(* IEC 61131-3 sources: Dev/Dev_V200/200 (part 4) *)

	   _229_S : UDINT := SIZEOF(NH_FRM_229); _229 : NH_FRM_229;
   	_230_S : UDINT := SIZEOF(NH_FRM_230); _230 : NH_FRM_230;
	   _231_S : UDINT := SIZEOF(NH_FRM_231); _231 : NH_FRM_231;
		_232_S : UDINT :=	SIZEOF(NH_FRM_232); _232 : NH_FRM_232;
		_233_S : UDINT :=	SIZEOF(NH_FRM_233); _233 : NH_FRM_233;
		_234_S : UDINT :=	SIZEOF(NH_FRM_234); _234 : NH_FRM_234;
		_235_S : UDINT :=	SIZEOF(NH_FRM_235); _235 : NH_FRM_235;
		_236_S : UDINT :=	SIZEOF(NH_FRM_236); _236 : NH_FRM_236;

		_246_S : UDINT :=	SIZEOF(NH_FRM_246); _246 : NH_FRM_246;
	//	_247_S : UDINT :=	SIZEOF(NH_FRM_247); _247 : NH_FRM_247;
		_248_S : UDINT :=	SIZEOF(NH_FRM_248); _248 : NH_FRM_248;
	//	_249_S : UDINT :=	SIZEOF(NH_FRM_249); _249 : NH_FRM_249;
		_260_S : UDINT := SIZEOF(NH_FRM_260); _260 : NH_FRM_260 ;

(*
   _0_S : UDINT := SIZEOF(NH_FRM_0); _0 : NH_FRM_0 ;
   _0_S : UDINT := SIZEOF(NH_FRM_0); _0 : NH_FRM_0 ;
   _0_S : UDINT := SIZEOF(NH_FRM_0); _0 : NH_FRM_0 ;
*)

	   _END_FRM_WEB    : UDINT := 0;

	END_VAR

	FUNCTION_BLOCK _Nh_Create_FRM
   	VAR_INPUT
         Go          : USINT;
			all			: BOOL;
   	END_VAR
   	VAR_OUTPUT
         done        : BOOL;
			busy			: BOOL;
	      cyc         : UINT;
   	   files       : UINT;
      	actSize     : UDINT;
//         expTime    	: TIME;
   		GoNext		: USINT;
		END_VAR
   	done  := false;
      CASE go OF
       0 :  RETURN;
       1 :
            xFrmHed  := ADR(_START_FRM_SYS);
            Go 		:= 3;
				IF all THEN
					_Nh_Log_Path(wh:=21, frm:=1);
// 	           rb       := ForceDirs(fileName := yTx2);
					yTx2 		:= CONCAT('New FRM_SYS: ',yTx2);
 					rb 		:= _Nh1RowTxt(logRst := 1);
					GoNext   := 2;
   			ELSE
					GoNext   := 0;
				END_IF;
				all	:= false;
       2 :
      		GoNext	:= 0;
				{$IFDEF __NH_WEB}
					xFrmHed  := ADR(_START_FRM_WEB);
					_Nh_Log_Path(wh:=21, frm:=1);
					yTx2 		:= CONCAT('New FRM_WEB: ',yTx2);
 					rb 		:= _Nh1RowTxt(logRst := 1);

               Go    	:= 3;
            {$ELSE}
               Go    	:= 99;
   			{$END_IF}

       3 :
				busy		:= true;
            cyc      := 0;
            files    := 0;
            actSize  := 0;
            xFrmHed  := xFrmHed + 1;
            Go       := 4;

       4 :
      	   cyc   := cyc + 1;
				_Nh_Log_Path(wh:=21, frm:=1);
            WHILE xFrmHed^.Size > 0 DO
      	      yTx3 := CONCAT(yTx2, xFrmHed^.hed.Name ,'.FRM');
         	   fH   := FileOpen(fileName := yTx3, mode := F_WRITE);
            	IF fH <> INVALID_HANDLE_VALUE THEN
               	sz       := PTR_TO_UDINT(xFrmHed) + 4;
      	         sz       := FileWrite (hFile := fH, adrBuf := sz, size := xFrmHed^.size);
         	      actSize  := actSize + sz;
            	   files    := files + 1;
               	aSys.RWtoFileCycle := aSys.RWtoFileCycle + sz;
      	      END_IF;
         	   rb       := FileClose (hFile := fH);
      	      sz       := xFrmHed^.size + 4;
         	   xFrmHed  := xFrmHed + sz;
					IF _NhMaxRWLimit() OR _NhMaxTimeCyc()  THEN
						EXIT;
					END_IF;
(*
      	      expTime  := SUB_DT_DT(GetRTC(),aSys.NhDT);
      	      IF aSys.RWtoFileCycle > 32768 OR expTime > T#0.2s THEN
         	      EXIT;
            	END_IF;
*)
      	   END_WHILE;
         	IF xFrmHed^.Size = 0 THEN
               Go       := 99;
      	   END_IF;
       99:
				Go := GoNext;
				IF Go = 0 THEN
         	   Done := TRUE;
         	   Busy := false;
				END_IF;
      END_CASE;
	END_FUNCTION_BLOCK

	VAR_GLOBAL
   	fb_Nh_Create_FRM    : _Nh_Create_FRM;
	END_VAR

{ $ END_IF }

(* ---- _Nh_Het.st ---- *)
TYPE

(*
   NH_HET_DIS	{HIDDEN} :  STRUCT 		    // prenos medzi HET a TGL,WSB....
		ok 			: BOOL;                 	// mame ReQ teplotu z tohto regulatora
		chg			: BOOL;       				   // zmena ReQ
		valReQ		: REAL;                    // pozadovana velicina
		valAct		: REAL;                    // aktualna velicina
   END_STRUCT;
*)

END_TYPE

TYPE

END_TYPE

TYPE
END_TYPE

TYPE
END_TYPE

FUNCTION _Nh_PvValOut  {HIDDEN} : USINT		// nastavi vystupny stupen KURENIA/CHLADENIA podla hysterezie
	VAR_INPUT
   	het		: BOOL;
		up			: USINT;
		pv			: USINT;
		reQ		: REAL;
		val		: REAL;
		wht		: PTR_TO NH_HET_MODE;
  	END_VAR
//	vr	:= wht^.reQ[ pv ];
	i	:= 3;
	WHILE i >= 1 DO
		kr := wht^.hys[up,i];

(*
		IF up THEN
			kr		:= wht^.hys.up[i];
		ELSE
			kr		:= wht^.hys.dn[i];
		END_IF;
*)
		IF het THEN														// kurenie

(*
					UP                 		DN
			23.3  0.                      0.
			23.2  0.                      0.
			23.1  0.                 		1.	<= [23+0.1=23.1]
			23.0  0 --------------------- 1.
			22.9	0.                      2.	<= [23-0.1=22.9]
			22.8  0.                      2.
			22.7  0.                      2.
			22.6	0.	                     2.
			22.5  1.	<= [23-0.5=22.5]     2.
			22.4  1.                      2.
			22.3  1.                      3.	<= [23-0.7=22.3]
			22.2  1.                      3.
			22.1  1.                      3.
			22.0  2.	<= [23-1.0=22.0]     3.
			21.9  2.                      3.
			21.8  2.                      3.
			21.7  2.
			21.6  2.
			21.5  2.
			21.4  2.
			21.3  2.
			21.2  2.
			21.1  2.
			21.0  3.	<= [23-2.0=21.0]
			20.9	3.
*)

//			IF val <= reQ - kr THEN
			IF val <= reQ + kr THEN
				EXIT;
			END_IF;
		ELSIF	pv = 0 THEN												// pri chladenie/vetrani/odvlhceni je PV=0 OFF
			i := 1;
		ELSIF val >= reQ + kr THEN
			EXIT;
		END_IF;
		i := i-1;
	END_WHILE;
	_Nh_PvValOut := i;
END_FUNCTION

TYPE

END_TYPE

(* ---- _Nh_Ini.st ---- *)
(* INICIALIZACNE FUNKCIE RAM A DBX PO RESTARTE, OBNOVENIE Z SDC A TESTY KONZISTENCIE  *)
(*
TYPE
  	NH_DBX_2	{HIDDEN}   :  STRUCT 			// riadiaca hlavicka DBX
      ver         : NH_DBX_VER   ;
      sCfg        : USINT := SIZEOF(NH_CFG_CFG);       // velkost vety aCfg v DBX
      sPar        : USINT := SIZEOF(NH_PAR_CFG);       // velkost vety aPar v DBX
      sVaz        : USINT := SIZEOF(NH_VAZ_CFG);       // velkost vety aVaz v DBX

      nCfg        : USINT := _Nh_CFG;              // pocet viet CFG
      nPar        : USINT := _Nh_PAR;              // pocet viet PAR
      nVio        : USINT := _Nh_VAZ;              // pocet viet VAZ
      // adresy dat
      aCfg        : UINT;                          // offset od _Dbx0  - zaciatok aCfg ulozeny v databoxe
      aPar        : UINT;                          // zaciatok aPar ulozeny v databoxe
      aVio        : UINT;                          // zaciatok aVaz ulozeny v databoxe
      vRam        : UINT;                          // aktualna velkost dat v aRam[] = posladny zaznam aVaz
      // gobalne  premenne/sablony, ktore sa obnovuju z DBX
      all         : NH_DBX_VAR;
      rezerva     : STRING[79];
//    0,ROM,ZON,CAT,SCN,FAV,USR,HET,SVD,SVA,RGB,ZAS,STY,VEN,ROL,GAR,SIR,13,WSB,TLA,KOT,TVE,CER,PIR,TER,DOR,WIN,LUX,KEY,H20,FIR,GAS,
//      ixc         : ARRAY[0..50] OF USINT := [0,3,1,2,5,4,20,22,6,10,11,12,21,23,31,32,30,13,14,8,7,9,15,16,17,18,19,24,27,28,29,38,39,0]; // SCN,SVD,SVA....
//      ixc         : ARRAY[0..50] OF USINT := [0,1,3,4,5,20,22,10,11,12,21,23,31,32,33,34,35,30,13,14,24,15,19,16,17,18,6,7,8,9,27,28,29,37,38,39,2,0]; // SCN,SVD,SVA....
	END_STRUCT;

   NH_CFG_CFG_2  {HIDDEN}:  STRUCT 					// zakladny konfiguracny subor vsetkych DEV a ich rozlozenie v RAM
      // spoloxna struktura pre xNh
		Siz         : UDINT;								// velkost jedneho zaznamu
		Ram         : UDINT;							  // adresa 1.vety vo virtualnej pamati mRam[ vRam ], kde je ulozena xCfg (nulta veta )
      Rec         : INT;                       // pocet zaznamov
		New			: INT;						     // pocet novych zanamov, ktore sa ziadaju
      nDe         : USINT;                       // pocet DEL-viet
      rDe         : INT;                       // posledna volna DEL veta
      NOk         : BOOL;                      // novopridana veta bude oznacena uz pri pridani ako platna
      ver         : USINT := 1;
		// dotial musia mut CFG,PAR,VAZ rovnake, kebo sa pouzivaju xNh^
  		cfg			: STRING[3] ;						// nazov suboru na SDC dev := xxx.***
      ofs         : UDINT;                       // offset Empty premennej od eRom
      // unikatne  pre CFG
      par         : USINT;                      // cislo parametra  (odkaz do aPar)
      al          : USINT;	// := SIZEOF(NH_DEV_ALL) ;                      // velkost specialnej cfg pre dev
      cx          : USINT;                      // velkost specialnej cfg pre dev
      // dotialto sa obnovuje DBXver=001
      cf          : USINT := SIZEOF(NH_CFG_ALL);                      // velkost hlavnej cfg
      me          : UINT;                       // velkost uzivatelskej prevadzkovej pamate
      hw          : USINT;                       // velkost HW pamate
      io      		: USINT;
      dummy5      : USINT;
      dummy6      : USINT;
      dummy7      : USINT;
      dummy8      : USINT;
      dummy9      : USINT;
      // dotialto sa obnovuje DBXver > 001
      cat         : USINT;                      // cislo cat do ktorej patri toto dev
      ref         : USINT := 251;               // druh refreshu 251-len to co je na obrazovke,252=to co je na obrazevke a predefinovat,254=novy vypis od 1.zanamu
//      cou         : USINT;                      // cislo skupiny vystupov pre prenos vstupov
      tgr         : USINT;                      // typovy predstavitel/skupina vazieb

      mna         : USINT;                      // cislo menu pre ikonu vlastnosti - administrator _042.MN0
      mnu         : USINT;                      // cislo menu pre ikonu vlastnosti - user          _042.MN0
      rExp        : USINT;                      // pocet viet v z exportu
      fBr         : USINT;                      // cislo formatoveho suboru pre pre BRW-ROW, ulozene _Nh_ADR_ROT,'/CFG/FRM/_000.
      fSc         : USINT := 200;               // cislo menu cez ktore sa dostane so _Nh_Frm_SCR = parametrov DEV
      ar2         : BOOL;                       // '>>' dvojita      sipka dalej je v obr[4] prioritou c.1
      lst         : BOOL;                       // ma ikonu DEV-listu {SCN,ACT..}
      stp         : BOOL := true;               // moze mat odskok na vazby = ikona setup (len v rezime setup)
      fav         : BOOL := true;               // ma ikonu fav
      chk         : BOOL := true;               // ma ikonu check (ak je vo vazbach)
      edn         : BOOL := true;               // moze sa editovat nazov
      sld         : BOOL;                       // DEv ma slider v riadkovom zobrazeni
      ou          : BOOL;                       // tot je vystup - kde sa nieco nastavuje
      dbx         : BOOL;                       // data boli obnovene z DBX
      sdc         : BOOL;                       // data boli obnovene z SDC
//      NoDelDBX    : BOOL;                       // pri obnoveni z DBX sa NE-oznaci ako DEL. Potom ju odznaci proces aktualizacie adries z NH2.ADR
      NoRecCat    : BOOL;                       // pri zfiltrovani kategorie sa zobrazia aj ked nemaju ziadny zaznam
      AllCFG      : BOOL;                       // z DBX neobnovuje po cf+al+cx... ale obnovi naraz cely zaznam podls velkosti SIZE
      scn         : BOOL;                       // priznak, ze ide o dev, ktore riadi viac vystupnych DEV (SCN,ACT,TIM...)  ma nejeky dev-list
      body        : BOOL;                       // tento DEV zapisuje pritomnost
      ini         : BOOL;                       // pri inicializacii boli pridane vety, treba ich popisat
      del         : BOOL;			               // je mozne mazat DEV (ON/OFF)
      bck         : BOOL := true;               // toto cfg sa zalohuje z RAM -> SDC
      imp         : BOOL := true;               // do cf sa importuju adresy  z CIB .... , ROM nebude mat adresy
      NewExp      : BOOL;                       // toto CFG ma z exportu nove data/adresy a musi sa aktualizovat
      QckStat     : BOOL;                       // v HOME-QuickMnu sa vypisuju obrazku zo stat, nie z dev
      lvl254      : BOOL;                       // dev nema max LVL 100% ale 254 = DALI            (len pre web)
      analog      : BOOL;                       // dev je 0-100% alebo 0-254                       (len pre web)
      dali      	: BOOL;                       // patri do dali
      ShwSta   	: BOOL;  		              // robrazi sa ikona cfg v ROM/ZON ak je niektore z DEV v [cf] aktivne
      zone        : BOOL;                       // moze vstupovat {davat signal} aj do zony  (TER,LUX)

   END_STRUCT;

  	NH_PAR_CFG_2  {HIDDEN}:  STRUCT 					// zakladny konfiguracny subor vsetkych parametrov
      // spoloxna struktura pre xNh
		Siz         : UDINT;								// velkost jedneho zaznamu
		Ram         : UDINT;							  // adresa 1.vety vo virtualnej pamati mRam[ vRam ], kde je ulozena xCfg (nulta veta )
      Rec         : INT;                       // pocet zaznamov
		New			: INT;						     // pocet novych zanamov, ktore sa ziadaju
      nDe         : USINT;                       // pocet DEL-viet
      rDe         : INT;                       // posledna volna DEL veta
      NOk         : BOOL;                      // novopridana veta bude oznacena uz pri pridani ako platna
      ver         : USINT := 1;

		cfg			: STRING[3] ;						// nazov suboru na SDC dev := xxx.***
      ofs         : UINT;                       // offset Empty premennej od epSvd

      // unikatne  pre PAR
      dbx         : BOOL;                       // data boli obnovene z DBX
      sdc         : BOOL;                       // data boli obnovene z SDC
//		in          : BOOL := true;					//	vo vazbe IN sa vytvara parameter, inak sa preberie z hlavicky
//		ou          : BOOL := true;					// vo vazbe OU sa vytvara parameter, inak sa preberie z hlavicky
      grp         : BOOL;                       // novy parameter sa vytvori, len ak vstupuje na pozici OUT skupinovych prikazov do SCN,ACT,TIM. Inak sa zoberie default cislo paramtra z DEV
//		New			: INT;						     // pocet novych zanamov, ktore sa ziadaju
	END_STRUCT;

  	NH_VIO_CFG_2	{HIDDEN}   :  STRUCT 			  // zakladny konfiguracny subor vazieb
		Siz         : UDINT := SIZEOF(NH_VAZ);	  // velkost jedneho zaznamu
		Ram         : UDINT;							  // adresa 1.vety vo virtualnej pamati mRam[ vRam ], kde je ulozena xCfg (nulta veta )
      Rec         : INT;                       // pocet zaznamov
		New			: INT;						     // pocet novych zanamov, ktore sa ziadaju
      nDe         : USINT;                       // pocet DEL-viet
      rDe         : INT;                       // posledna volna DEL veta
      NOk         : BOOL;                      // novopridana veta bude oznacena uz pri pridani ako platna
      ver         : USINT := 1;

      ref         : BOOL := true;              // vsetky vazby sa refreshnu (ako keby bolo cmd > 0)
	   ini         : BOOL;                      // pri restarte sa nplni DEFAULT hodnotami
   END_STRUCT;
END_TYPE

VAR_GLOBAL
	oDbx	      {HIDDEN}	   : NH_DBX_2;                                // hlavny riadiaci subor vratane organizacie DBX
   oCfg        {HIDDEN}    : NH_CFG_CFG_2;                            // konfiguracia vsetkych DEV
   oPar        {HIDDEN}    : NH_PAR_CFG_2;                            // konfiguracia vsetkych DEV
   oVio        {HIDDEN}    : NH_VIO_CFG_2;                            // konfiguracia vsetkych DEV
END_VAR
*)

VAR_GLOBAL CONSTANT
(*
  _NhQickGuide   {HIDDEN} : ARRAY[ 9..16,0..1] OF USINT :=
                    [   1,  0,                     // Vytvorit miestnost
                        2, 44,                     // Dev bezmiestnosti
                        2, 16,
                        2, 15,
                        2, 24,
                        2, 14,
                        2,  5,
                        2,  6
                    ];
END_VAR
*)

  _NhQickGuide   {HIDDEN} : ARRAY[ 9..14,0..1] OF USINT :=
                    [   2, 16,
                        2, 15,
                        2, 24,
                        2, 14,
                        2,  5,
                        2,  6
                    ];
END_VAR

FUNCTION _NhNewPAR {HIDDEN} : BOOL	    // zvysi poziadavku na novu vetu (vrati true), alebo oznaci existujucu ak je DEL (false)
   VAR_INPUT
      xP    : PTR_TO INT;                          // xCfg^.par, alebo io.p
      cp    : USINT;
		ee	: INT;
   END_VAR
   _NhNewPAR := true;                             // default nepridavaju sa nove vety

(*
	IF cp = 14 THEN
      yTx2     := CONCAT('  nd: ',INT_TO_STRING(nd), ' cp: ',USINT_TO_STRING(cp),' np: ',INT_TO_STRING(xP^)   );
      _Nh1RowTxt(logRst:=1, noTime := 1);

//		aSys.ini := 217;
//		RETURN;

	END_IF;
*)

   IF xP^ = 0	THEN																// nememe parameter a mal by byt
      ;
   ELSIF xP^ > aPar[cp].rec THEN                   // parameter sa este len prida, ale uz si ho nieco rezervovalo
		j := j+1;
	ELSIF _NhxPar(cp := cp, np := xP^ ,x:=ee) THEN   // uz si ho zobralo iny DEV, musi sa vytvoriy novy
		i := i + 1;
   ELSE
       _NhNewPAR   := false;                        // pridava sanew := true;
       xPar^.ok.ok := true;
		z := z + 1;
   END_IF;
   IF _NhNewPAR THEN
      aPar[cp].new   := aPar[cp].new + 1;
      aPar[cp].nOk   := true;                                        // pridane vety budu hned platne
      xP^            := aPar[cp].rec + aPar[cp].new;   // parametrom bude nova platna veta
		x				 	:= x + 1;
   END_IF;
(*
	IF cp = 14 THEN
      yTx2     := CONCAT('    j: ',SINT_TO_STRING(j), ' i:',USINT_TO_STRING(i), ' z:',INT_TO_STRING(z),' x:',INT_TO_STRING(x)   );
      _Nh1RowTxt(logRst:=1, noTime := 1);
	END_IF;
*)

END_FUNCTION

FUNCTION _Nh_Ini_PAR_Test {HIDDEN}   : BOOL	    // prejde vsetky DEV, ktore maju parametre a tieto parametre prida,a lebo od-DELETUJE
   VAR_TEMP
      cp       : USINT;
   END_VAR
   IF aSys.exp = 0 THEN
      yTx2     := 'START - _Nh_Ini_PAR_Test KONTROLA PARAMETROV :';
      _Nh1RowTxt(logRst:=1);
   END_IF;
   aSys.exp := aSys.exp + 1;
   WHILE aSys.exp <= aDbx.nCfx[0] DO                                       // prechadzaju sa typy parametrov kazdom cykle
      IF aCfg[aSys.exp].par = 0  THEN                                          // nema cf typ CFG_ALL, a tym ani parametre
         RETURN;
      END_IF;

	x	:= 0;
	y	:= 0;
	z	:= 0;
	i	:= 0;
	j	:= 0;

      cp    := aCfg[aSys.exp].par;
      FOR nd := 1 TO aCfg[ aSys.exp ].rec DO                         // prechadza len toto cfg
			IF _NhxPt( c := aSys.exp, n := nd, x:=70) OR aCfg[aSys.exp].dali THEN           // testuje len platne vety,
				IF cp = 0 THEN
               IF xPt^.cf.par > 0 THEN
						xPt^.cf.par	:= 0;                                    // grp je len pre ACT,SCN
						y				:= y + 1;
					END_IF;
				ELSE
				   _NhNewPAR(cp := cp, xP := ADR(xPt^.cf.par), ee:=60);
				END_IF;
			END_IF;
    	END_FOR;
     	yTx2	:= '  ' +USINT_TO_STRINGF(aSys.exp,'%3d')
		  			+ ' ' + aCfg[ aSys.exp ].cfg
					+ ' Rec: ' + INT_TO_STRINGF(aCfg[aSys.exp].rec,'%3d')
					+ ' Del: ' + INT_TO_STRINGF(y,'%3d');

		IF cp > 0 THEN
	     	yTx2	:= yTx2
						+ ' Ok: '  + INT_TO_STRINGF(z,'%3d')
						+ ' New: ' + INT_TO_STRINGF(x,'%3d')
		  				+ ' ' + aPar[cp].cfg
						+ ' ' + INT_TO_STRINGF(aPar[cp].rec,'%3d')
						+ ' D: ' + USINT_TO_STRINGF(i,'%3d');
		END_IF;
		IF aCfg[ aSys.exp ].cfg <> '' THEN
	  		rb       := _Nh1RowTxt(logRst := 1);
		END_IF;
		IF x > 0 THEN
			_Nh_Go_DbxToMem(ram := true,dbx := false );                        // zalozi RAM->DBX, z DBX vrati do RAM s pridanim novych uz platnych viet
		END_IF;

      RETURN;
   END_WHILE;
   aSys.ini := 214;
   yTx2     := CONCAT('END - Kontola PAR Ok. aSys.ini:=', USINT_TO_STRING(aSys.ini) );
   rb       := _Nh1RowTxt(logRst := 1);
END_FUNCTION

FUNCTION _NhIniVAZ  {HIDDEN} : BOOL	    // prejde vazby a ak v IN alebo OUT je DEV, ktore neexistuje, vymaze vazbu
   VAR
      nvz    : USINT;
//      io    : USINT;
//      chg   : INT;
//      old   : INT;
      par   : INT;
      ndv   : INT;
      cp       : USINT;
   END_VAR
	yTx2     := '_NhIniVAZ     : ZACINAM KONTROLU';
 	_Nh1RowTxt(logRst:=1);

	FOR nvz := 2 TO 4 DO
		x	:= 0;
		y	:= 0;
		z	:= 0;
		i	:= 0;
		FOR ndv := 1 TO aVaz[nvz].Rec DO
         IF _NhxVaz( cv := nvz, nd := ndv) THEN                             // veta vazby je platna
				ok	:= true;

		  		IF _NhxPt(c:=xVaz^.in.c,n:=xVaz^.in.n,err:=1 ,x:=22) = false THEN
					xVaz^.ok.ok 	:= false;
					ok	   			:= false;
				ELSIF _NhxPt(c:=xVaz^.ou.c,n:=xVaz^.ou.n, err:=1 ,x:=24) = false THEN
					xVaz^.ok.ok 	:= false;
					ok	   			:= false;
				END_IF;

				IF ok THEN
					cp := aCfg[xVaz^.in.c].par;
					IF nvz = 3 THEN
						cp := 0;
					END_IF;
					IF cp = 0 THEN
						IF xVaz^.in.p > 0 THEN
							xVaz^.in.p := 0;
							y			  := y + 1;
						END_IF;
					ELSIF xVaz^.in.p > 0 THEN
					   _NhNewPAR(cp := cp, xP := ADR(xVaz^.in.p), ee:=61);
					END_IF;
					cp := aCfg[xVaz^.OU.c].par;
					IF cp = 0 THEN
							IF xVaz^.OU.p > 0 THEN
							xVaz^.OU.p := 0;
							y			  := y + 1;
						END_IF;
					ELSIF xVaz^.OU.p > 0 THEN
				   	_NhNewPAR(cp := cp, xP := ADR(xVaz^.OU.p), ee:=62);
					END_IF;
	         END_IF;
			END_IF;
      END_FOR;
     	yTx2	:= '   ' + USINT_TO_STRING(nvz)
		  			+ ': Rec: ' + INT_TO_STRINGF(aVaz[nvz].rec,'%3d')
					+ ' Del: ' + INT_TO_STRINGF(y,'%3d')
					+ ' Ok: '  + INT_TO_STRINGF(z,'%3d')
					+ ' New: ' + INT_TO_STRINGF(x,'%3d')
					+ ' Dupl: ' + USINT_TO_STRINGF(i,'%3d');
 		rb       := _Nh1RowTxt(logRst := 1);
		IF x > 0 THEN
			_Nh_Go_DbxToMem(RAM := true,dbx := false );                        // zalozi RAM->DBX, z DBX vrati do RAM s pridanim novych uz platnych viet
		END_IF;
	END_FOR;

	yTx2     := '_NhIniVAZ     : KONTROLA OK.';
 	_Nh1RowTxt(logRst:=1);

END_FUNCTION

FUNCTION _Nh_Ini_Default_CFG_INI {HIDDEN}    : BOOL	    // doplni default CFG, ak este nie je
	VAR_INPUT
		vz		: BOOL;
		ver	: BOOL := true;
		nOk	: BOOL := true;
		rec	: INT;
		cf		: USINT;
	END_VAR
   _Nh_Ini_Default_CFG_INI := false;                             // default nepridavaju sa nove vety
	IF vz	THEN
	   IF aVaz[cf].rec < rec  THEN   // ver=0: FAV,USR
   	   IF aVaz[cf].rec < rec THEN
      	   aVaz[cf].new :=  rec  - aVaz[cf].rec ;
	      END_IF;
   	   aVaz[cf].ini := TRUE;
      	aVaz[cf].nOk := nOk;
   	END_IF;
	 	aCfg[cf].ini   := aVaz[cf].ini OR ver;
	ELSE
		IF rec > aCfg[cf].rec THEN                                         // porovna sa aktulny pocet s pozadovanym
 			aCfg[cf].nOk	:= nOk;
	      aCfg[cf].new   := rec  - aCfg[cf].rec ;
   	   aCfg[cf].ini   := true;                                        // do tohto CFG sa budu pridavat detault vety
   		yTx2 := CONCAT('..',aCfg[cf].cfg,' + ',INT_TO_STRING(aCfg[cf].new) );
			rb   := _Nh1RowTxt(logRst := 1);
		END_IF;
		IF ver AND aCfg[cf].ver = 0 THEN
		 	aCfg[cf].ini   := true;
		END_IF;
	END_IF;
END_FUNCTION

FUNCTION _Nh_Ini_Default_CFG_DEF {HIDDEN} : BOOL	    // nakopiruje default sablony
	VAR_INPUT
		cf		: USINT;
		frm	: UINT;
	END_VAR
   _Nh_Ini_Default_CFG_DEF := false;                             // default nepridavaju sa nove vety
	IF aCfg[cf].ini = false THEN                                         // porovna sa aktulny pocet s pozadovanym
		RETURN;
	END_IF;
	// cele preddefinovane sablony
 	_Nh_FRM_Read(frm:=frm);               // zone
	MemCpyEx (	length := aCfg[cf].siz * MIN( USINT_TO_UDINT(yFrmName.row), INT_TO_UDINT(aCfg[cf].rec)) ,
				source := VOID( yFrmData ), dest := VOID( mRam[ aCfg[cf].ram ] ));
END_FUNCTION

FUNCTION _Nh_Ini_DEFAUL_CFG  {HIDDEN}    : BOOL	    // doplni default CFG, ak este nie je
   VAR_TEMP
      dsh,
//      zon                     : BOOL;
//      _NhCrPOI                : BOOL;
//      w                       : INT;
      cf                      : USINT;
   END_VAR
   yTx2 	:= 'START-kontroly Default udajov {_Nh_Ini_Default_DEFAUL}';
   rb   	:= _Nh1RowTxt(logRst:=1);
	// pripravi pocet novych viet
	_Nh_Ini_Default_CFG_INI(cf:= 3,rec:=USINT_TO_INT(_NH_ZONES));   // ZON 1=domov,2=vnutro,3=vonku.  Ostatne xony sa musia pridat rucne
	_Nh_Ini_Default_CFG_INI(cf:=20,rec:=4);          					// FAV defult je 4
	_Nh_Ini_Default_CFG_INI(cf:=22,rec:=USINT_TO_INT(_Nh_USR));     // USR
	_Nh_Ini_Default_CFG_INI(cf:=25,rec:=1);      							// GLB
	_Nh_Ini_Default_CFG_INI(cf:=48,rec:=7);      							// ALA
	_Nh_Ini_Default_CFG_INI(vz:=true, cf:= 1,rec:=USINT_TO_INT(_Nh_USR)*8, ver:=aCfg[20].ver=0 OR aCfg[22].ver=0); // VAZ[1]
	{$IFDEF __NH_DALI}
   IF _Nh_DALI_MA > 0 THEN
		_Nh_Ini_Default_CFG_INI(cf:=42,rec:=USINT_TO_INT(_Nh_DALI_MA), nOk:=0);      				// DLM
		_Nh_Ini_Default_CFG_INI(cf:=43,rec:=USINT_TO_INT(_Nh_DALI_MA)*64);   				// DLS
		_Nh_Ini_Default_CFG_INI(cf:=44,rec:=USINT_TO_INT(_Nh_DALI_MA)*16);   				// DLG
   END_IF;
	{$END_IF}
	// nakopirovat sablony

	_Nh_Go_DbxToMem(dbx := false, ForceRamOk:=true);         	// ulozi MEM->DBX a spat nacita este raz z DBX a prida nove vety
	_Nh_Ini_Default_CFG_DEF(cf:= 3,frm:=252);     // ZON
	_Nh_Ini_Default_CFG_DEF(cf:=20,frm:=251);     // FAV
	_Nh_Ini_Default_CFG_DEF(cf:=22,frm:=253);     // USR
//	_Nh_Ini_Default_CFG_DEF(cf:=  ,frm:=254);		// MSG
	_Nh_Ini_Default_CFG_DEF(cf:=48,frm:=255);		// ALA

   // vytvori sadu HOME-DSH pre kazeho usra
   cf := 1;
// aVaz[1].ini := 1;
   IF aVaz[1].ini THEN
		_Nh_FRM_Read(frm:=250);
		sz		:= aVaz[1].ram;
		sp		:= SIZEOF(NH_VAZ) * 8;
      FOR i := 1 TO _Nh_USR DO
         _NhxUsr(u := i );
         // fac.c je cislo usra 1..5
         xUsr^.cx.fav.c   := 1; xUsr^.cx.fav.n   := 0;            // FAV je spolocny pre vsetkych
         xUsr^.cx.dsh.c   := i;
         xUsr^.cx.qck.c   := i;
         xUsr^.cx.ds1     := xVaz^.ou;                           // cislo preveho DEV v DSH cf/nd
			FOR ii := 1 TO 8 DO
				yFrm_250.vz1[ii].in.c := i;
         END_FOR;
			MemCpyEx (	length := sp ,
							source := VOID( yFrmData ), dest := VOID( mRam[ sz ] ));

			sz	:= sz + sp;
		END_FOR;

(*

      xVaz  := ADR(mRam[aVaz[cf].ram]);
      sPtr  := aVaz[cf].Siz;
      // vycisti vsetok FVL (vazby)
      memset(val := 0, length := INT_TO_UINT(aVaz[cf].rec) * UDINT_TO_UINT(sPtr), dest := VOID( mRam[ aVaz[cf].ram ] ));
      // ku kazdemu usrovy dokopiruje sadu DSH 1..8 a u USR nastavi FAV na spolocny (c:=1,n:=0)
      FOR i := 1 TO _Nh_USR DO
         // nakopiruje 8 viet DSH
//         _Nh_FRM_Read(wht:=251, frm:=250, cfg:=1, sz := 8 * sPtr , ofs := 8 * sPtr * USINT_TO_UDINT(i-1) );
         _Nh_FRM_Read(frm:=250);
         _NhxUsr(u := i );
         // fac.c je cislo usra 1..5
         xUsr^.cx.fav.c   := 1; xUsr^.cx.fav.n   := 0;            // FAV je spolocny pre vsetkych
         xUsr^.cx.dsh.c   := i;
         xUsr^.cx.qck.c   := i;
         xUsr^.cx.ds1     := xVaz^.ou;                           // cislo preveho DEV v DSH cf/nd
         FOR nd := 1 TO 8 DO
            xVaz^.in.c  := i;                                     // preznaci usra u nakopitovanej sady
            xVaz        := xVaz + sPtr;
         END_FOR;
      END_FOR;
*)
   END_IF;
END_FUNCTION

(*
FUNCTION _Nh_Ini_Default_DEFAUL    : BOOL	    // doplni default CFG, ak este nie je
   VAR_TEMP
      ok,dsh,usr,sbj,
      zon                     : BOOL;
      _NhCrPOI                : BOOL;
      w                       : INT;
      cf                      : USINT;
   END_VAR
   yTx2 := 'START-kontroly Default udajov {_Nh_Ini_Default_DEFAUL}';
   rb   := _Nh1RowTxt(logRst:=1);
   ok := false;

   // kontrola na DEFAULT vety v CFG (pocet)
   FOR cf := 1 TO _Nh_CFG DO
      xNh      := ADR(aCfg[cf]);
      ok1      := true;                                                 // default priznak, ze pridane vety budu hned OK
      CASE cf OF                                                        // CFG s minimalnym poctom viet. pridane vety budu hned oznacene ako OK
         3: ix := USINT_TO_INT(_NH_ZONES);                              // ZON 1=domov,2=vnutro,3=vonku.  Ostatne xony sa musia pridat rucne
        20: ix := 4;                                                    // FAV defult je 4
        22: ix := USINT_TO_INT(_Nh_USR);                                // USR defult je 5
        25: ix := 1;    																// GLB
      ELSE
         ix       := 0;
         ok1      := false;
      END_CASE;
      IF ix > aCfg[cf].rec THEN                                         // porovna sa aktulny pocet s pozadovanym
         xNh^.nOk       := ok1;
         aCfg[cf].new   := ix  - aCfg[cf].rec ;
         aCfg[cf].ini   := true;                                        // do tohto CFG sa budu pridavat detault vety
         ok             := true;                                        // globalny priznak, ze aspon do jedneho CFG treba pridat default vety
		   yTx2 := CONCAT('..',aCfg[cf].cfg,' + ',INT_TO_STRING(aCfg[cf].new) );
		   rb   := _Nh1RowTxt(logRst := 1);
      END_IF;
   END_FOR;

   cf:=1;   // FAV,FVL  - zoznam DSH pre kazdeho usra
   ix := USINT_TO_INT(_Nh_USR)*8;													// kazdy user ma 8 vlastnych Dash
   IF aVaz[cf].rec < ix OR aCfg[20].ver = 0 OR aCfg[22].ver = 0 THEN   // ver=0: FAV,USR
      IF aVaz[cf].rec < ix THEN
         aVaz[cf].new :=  ix  - aVaz[cf].rec ;
      END_IF;
      aVaz[cf].ini := TRUE;
      aVaz[cf].nOk := true;
      ok           := true;
   END_IF;
   cf             := 48;                                                            // ALArm
   aCfg[cf].ini   := true;
   ix := 7;
   IF ix > aCfg[cf].rec OR aCfg[cf].ver = 0 THEN    // novy ZON alebo POI
      If ix > aCfg[cf].rec THEN
         aCfg[cf].new   :=  ix  - aCfg[cf].rec ;
         aCfg[cf].nOk   := true;
         ok             := true;
      END_IF;
   END_IF;

	{$IFDEF __NH_DALI}
   IF _Nh_DALI_MA > 0 THEN
		ix	:= USINT_TO_INT(_Nh_DALI_MA);
	   IF aCfg[42].rec < ix THEN
	      aCfg[42].new := ix - aCfg[42].rec;
			ok 				:= 1;
			aCfg[42].NOk 	:= true;
   	END_IF;

		ix	:= USINT_TO_INT(_Nh_DALI_MA) * 64;
	   IF aCfg[43].rec < ix THEN
	      aCfg[43].new := ix - aCfg[43].rec;
			ok := 1;
   	END_IF;
		ix	:= USINT_TO_INT(_Nh_DALI_MA) * 16;
	   IF aCfg[44].rec < ix THEN
	      aCfg[44].new := ix - aCfg[43].rec;
			ok 				:= 1;
			aCfg[44].NOk 	:= true;
   	END_IF;
   END_IF;
	{$END_IF}

   IF ok THEN
      _Nh_Go_DbxToMem(dbx := false);                                 // len nacita este raz z DBX a prida nove vety
      FOR cf := 1 TO _Nh_CFG DO
         IF aCfg[cf].ini THEN                                     // tu je malo DEFAULT viet
            _NhxPt( c:= cf, n := 1,x:=52);                                     // prva veta
            CASE cf OF
               3: _Nh_FRM_Read(frm:=252);               // zone

RETURN;
              20: _Nh_FRM_Read(frm:=251);               // FAV - hlavicky
              22: _Nh_FRM_Read(frm:=253);               // users
              43: ;
//              46: _Nh_FRM_Read(wht:=250, frm:=254, cfg:=cf);               // MSG
              48: _Nh_FRM_Read(frm:=255);               // ALA
            END_CASE;
         END_IF;
      END_FOR;
   END_IF;

   // vytvori sadu HOME-DSH pre kazeho usra
   cf := 1;
// aVaz[1].ini := 1;
   IF aVaz[1].ini THEN
      xVaz  := ADR(mRam[aVaz[cf].ram]);
      sPtr  := aVaz[cf].Siz;
      // vycisti vsetok FVL (vazby)
      memset(val := 0, length := INT_TO_UINT(aVaz[cf].rec) * UDINT_TO_UINT(sPtr), dest := VOID( mRam[ aVaz[cf].ram ] ));
      // ku kazdemu usrovy dokopiruje sadu DSH 1..8 a u USR nastavi FAV na spolocny (c:=1,n:=0)
      FOR i := 1 TO _Nh_USR DO
         // nakopiruje 8 viet DSH
//         _Nh_FRM_Read(wht:=251, frm:=250, cfg:=1, sz := 8 * sPtr , ofs := 8 * sPtr * USINT_TO_UDINT(i-1) );
         _Nh_FRM_Read(frm:=250);
         _NhxUsr(u := i );
         // fac.c je cislo usra 1..5
         xUsr^.cx.fav.c   := 1; xUsr^.cx.fav.n   := 0;            // FAV je spolocny pre vsetkych
         xUsr^.cx.dsh.c   := i;
         xUsr^.cx.qck.c   := i;
         xUsr^.cx.ds1     := xVaz^.ou;                           // cislo preveho DEV v DSH cf/nd
         FOR nd := 1 TO 8 DO
            xVaz^.in.c  := i;                                     // preznaci usra u nakopitovanej sady
            xVaz        := xVaz + sPtr;
         END_FOR;
      END_FOR;
   END_IF;
END_FUNCTION
*)

FUNCTION _Nh_POI_INI {HIDDEN}   : BOOL	    // urobi testy POI, prida nove, vymaze stare
   // POI
	// 23.4.24
	ix					:= 0;
	aCfg[26].ini 	:= aCfg[26].ver = 0 ; // OR (aCfg[cf].ver = 2 AND aCfg[cf].ver_dbx < 2 );	// konverzia je 1 -> 2
   yTx2  			:= 'START - _Nh_POI_INI';
	_Nh1RowTxt(logRst:=1);

	ix := _Nh_POI_INI_REC();
   If ix > aCfg[26].rec THEN
      aCfg[26].new   := ix  - aCfg[26].rec ;
		aCfg[26].nOk 	:= false;
	   yTx2  := CONCAT('..Pridane aCfg[26].new : ',INT_TO_STRING(aCfg[26].new))  ;
		_Nh1RowTxt(logRst:=1);
      _Nh_Go_DbxToMem(ram:=true, dbx:=false);                                 		// len nacita este raz z DBX a prida nove vety
	ELSE
	   yTx2  := CONCAT('.._Nh_POI_INI - Ok. Rec: ',INT_TO_STRING(aCfg[26].rec))  ;
		_Nh1RowTxt(logRst:=1);
   END_IF;

	_Nh_POI_INI_NEW(cf:=  3, del := true);								// z ZON vzdy len vymaze poi
	IF aCfg[26].ini THEN
		// vsetky vety POI vymazat
	   yTx2  := CONCAT('.._Nh_POI_INI - DELETE  aCfg[26].rec : ',INT_TO_STRING(aCfg[26].rec))  ;
		_Nh1RowTxt(logRst:=1);
	   FOR ix := 1 TO aCfg[26].rec DO
			_NhxPt(ok:=1, c := 26, n := ix, x:=-123);             // najde aj del vetu
			xPt^.ok.ok := false;                          			// odznaci POI
		END_FOR;
		// najskor sa musi vymazat obsah - odkaz na poi v ROM,HET,HEV - VSETKO v jednom cykle CFG 1..X
		FOR cf := 1 TO _Nh_CFG DO
			IF aCfg[cf].NbrPoi > 0 THEN
		   	yTx2  := CONCAT('.._Nh_POI_INI - DEL-poi[day]: ',aCfg[cf].cfg,' ver:',USINT_TO_STRINGF(aCfg[cf].ver,'%3d') )  ;
				_Nh1RowTxt(logRst:=1);
				_Nh_POI_INI_NEW(cf:=cf, del:=true);				// vymazat NEW,DEL ROM/HET/HEV
			END_IF;
		END_FOR;
	END_IF;
	// teraz sa skontroluju odkazy POI, bud sa pridanaju alebo sa priradia
	FOR cf := 1 TO _Nh_CFG DO
		IF aCfg[cf].NbrPoi > 0 THEN
	   	yTx2  := CONCAT('.._Nh_POI_INI - CHK-poi[day]: ',aCfg[cf].cfg,' ver:',USINT_TO_STRINGF(aCfg[cf].ver,'%3d') )  ;
			_Nh1RowTxt(logRst:=1);
			_Nh_POI_INI_NEW(cf:=cf);				// kontrola, NEW,DEL ROM/HET/HEV
		END_IF;
	END_FOR;
   yTx2  := 'END -_Nh_POI_INI';
	_Nh1RowTxt(logRst:=1);
END_FUNCTION

FUNCTION _Nh_Ini_DEV_Test  {HIDDEN}  : BOOL	    // urobi testy
      cf := 1;
      FOR nd := 1 TO aCfg[1].rec DO
         IF _NhxPt(c:=cf, n:=nd) AND xPt^.cf.typ = 0 THEN
            _NhDefRom := INT_TO_USINT(nd);
            EXIT;
         END_IF;
      END_FOR;
      _Nh_Ini_DEV_Test := true;
      ix    := 1;                                                           		// presunie sa na dalsie CFG
      cf    := _Nh_IxC[ix];                                                     	// vybrate CFG
      WHILE  cf > 0 DO                                                           // prechadza zaznamy jedneho CFG
         nd    := 1;
         WHILE  nd  <= aCfg[cf].Rec DO                                           // vsetky vety CFG
            IF _NhxPt(c := cf, n := nd,x:=53) THEN
               xDev  := xPt;
					IF aCfg[cf].body THEN
						xDev^.cf.psn := true;                                          // len docasne do 5.9.23
   				END_IF;
//               IF cf = 23 THEN //   ú xDev^.cf.cat = 0 AND aCfg[cf].cat > 0 THEN
//               IF aCfg[cf].cat > 0 AND (xDev^.cf.cat = 0 OR xDev^.cf.cat <> aCfg[cf].cat) THEN
               IF cf = 4 THEN            														// sceny
                  xDev^.cf.cat := 53;                            						// default categoria
               ELSIF cf = 44 THEN            												// DLG
                  xDev^.cf.cat := 54;
               ELSIF aCfg[cf].cat > 0 AND (xDev^.cf.cat = 0 OR xDev^.cf.cat > _Nh_CAT) THEN
                  xDev^.cf.cat := aCfg[cf].cat;                            		// default categoria
               END_IF;

               IF cf = 1 THEN
						_Nh_TST_ROM();
					ELSIF cf = 3 THEN                                       				// zone ma ROM = nd
						_Nh_TST_ZON();
					ELSIF aCfg[cf].tgrp = 5 THEN                           				// ACT,ALA
                  IF xDev^.cf.rom = 0 OR xDev^.cf.rom > INT_TO_USINT(aCfg[3].rec) THEN      // kontrola na zone
                     xDev^.cf.rom := _NhDefHom; 														// domcek
                  END_IF;
					ELSIF xDev^.cf.rom = 0 THEN                                       // ostatne ako ROM nastavi na DEFault
     					xDev^.cf.rom := _NhDefRom;
               END_IF;
            END_IF;
            nd := nd + 1;
         END_WHILE;
         ix    := ix + 1;                                                           // presunie sa na dalsie CFG
         cf    := _Nh_IxC[ix];                                                     // vybrate CFG
      END_WHILE;

END_FUNCTION

{ $IFDEF __NH_EXP2 }

VAR_GLOBAL
	yWSBx	: NH_WSB;
	yTxXa	: STRING[255];
	yTxXb	: STRING[255];
END_VAR

{ $ END_IF  }
